PROGRAM P30_ManualControl
VAR
	i 	: INT;
END_VAR

FOR i:=1 TO 26 DO
	IF GVL_IO.aMaxValueController[i] <> 0 THEN
		GVL_IO.aController[i].nRampTime := GVL_IO.aController_RampTime[i];
		GVL_IO.aController[i].rTargetValue := GVL_IO.aController_TV[i] / GVL_IO.aMaxValueController[i] * GVL_IO.KL3464MaxValueH; //Input Set Value
		GVL_IO.aAnalogOutputIO[i] := LREAL_TO_INT(GVL_IO.aController[i].rControlValue); //Write to Device
		
		GVL_IO.aController_PV[i] := GVL_IO.aAnalogInputIO[i] / (GVL_IO.KL3464MaxValueH * GVL_IO.aMaxValueController[i]);
		GVL_IO.aController_CV[i] := LREAL_TO_REAL((GVL_IO.aController[i].rControlValue / GVL_IO.KL3464MaxValueH)*GVL_IO.aMaxValueController[i]);
		GVL_IO.aController[i]();
	END_IF
END_FOR


IF ( GVL_IO.aController_CV[27] > 10 ) THEN
// 		P11_E3508.bHeaterOn := TRUE;
	GVL_IO.aDigitalOutputIO[2].0 := TRUE;
ELSE
// 		P11_E3508.bHeaterOn := FALSE;
	GVL_IO.aDigitalOutputIO[2].0 := FALSE;
END_IF

GVL_IO.aController[27].nRampTime := GVL_IO.aController_RampTime[27];
GVL_IO.aController[27].rTargetValue := GVL_IO.aController_TV[27];
GVL_IO.wE3508_CV := LREAL_TO_WORD(GVL_IO.aController[27].rControlValue); //Write to Temperature Controller

GVL_IO.aController_PV[27] := WORD_TO_REAL(GVL_IO.wE3508_PV);
GVL_IO.aController_CV[27] := WORD_TO_REAL(GVL_IO.wE3508_CV);
GVL_IO.aController[27]();
				
(* Reactor Pressure Control *)
IF (GVL_IO.aController_TV[28] >= 0 ) THEN
	GVL_IO.aController[28].nRampTime := GVL_IO.aController_RampTime[28];
	GVL_IO.aController[28].rTargetValue := GVL_IO.aController_TV[28];
	GVL_IO.wIqPlus_CV := LREAL_TO_WORD(GVL_IO.aController[28].rControlValue); //Write to Pressure Controller
	
	GVL_IO.aController_PV[28] := WORD_TO_REAL(GVL_IO.wIqPlus_CDG2_PV);
	GVL_IO.aController_CV[28] := WORD_TO_REAL(GVL_IO.wIqPlus_CV);
	GVL_IO.aController[28]();
END_IF



(* Suceptor Rotation Control *)				
IF (GVL_IO.aController_TV[29] >= 0 ) THEN
	GVL_IO.aController[29].nRampTime := GVL_IO.aController_RampTime[29];
	GVL_IO.aController[29].rTargetValue := GVL_IO.aController_TV[29];
	GVL_IO.rRotation_ControlValue := LREAL_TO_REAL(GVL_IO.aController[29].rControlValue); //Write to Rotation Controller (rpm)
	
	GVL_IO.aController_PV[29] := GVL_IO.nRotation_Converted_PV;
	GVL_IO.aController_CV[29] := GVL_IO.rRotation_ControlValue;
	GVL_IO.aController[29]();	
END_IF

END_PROGRAM

(* stored: Version 1.1.0.1, ProductVersion 3.1.4026.11
   POU P30_ManualControl: Id {98ee4f4f-99e9-426e-9dfa-55ddf51d552b}, SpecialFunc None *)
